// TIA Portal V16 export
// export: Created 2021-11-12T13:31:11.6824383Z, ExportSetting WithDefaults, DisplayName Totally Integrated Automation Portal, DisplayVersion V16 Update 3, DisplayName TIA Portal Version Control Interface, DisplayVersion V16 Update 2, DisplayName TIA Portal Openness, DisplayVersion V16 Update 3, DisplayName SINAMICS Startdrive Advanced, DisplayVersion V16 Update 5, DisplayName SINAMICS Startdrive G130, G150, S120, S150, SINAMICS MV, S210, DisplayVersion V16 Update 5, DisplayName SINAMICS Startdrive G110M, G120, G120C, G120D, G120P, G115D, DisplayVersion V16 Update 5, DisplayName STEP 7 Professional, DisplayVersion V16 Update 3, DisplayName STEP 7 Safety, DisplayVersion V16, DisplayName WinCC UA Professional, DisplayVersion V16 Update 3
DATA_BLOCK "IDB_Sfty_Outputs"   // DB163, F_DB
{ DB_Accessible_From_OPC_UA := 'FALSE' }
VERSION : 0.1
// stored: AutoNumber true, DBAccessibleFromOPCUA false, InstanceOfName Sfty_Outputs, InstanceOfType FB
"Sfty_Outputs"
   // VAR
   //    "SF_100UH01-KF51_A1" : FDBACK;
   //    "SF_400UH01-KF51_A1" : FDBACK;
   //    "SF_100UH01-KF52_A1" : FDBACK;
   //    "SF_100UH01-KF53_A1" : FDBACK;
   // END_VAR
BEGIN
END_DATA_BLOCK
